// Mitsubishi GX Works2 project: PROG_ESTEIRA   PLC: Q03UDV
// PROG_ESTEIRA

PROGRAM MAIN
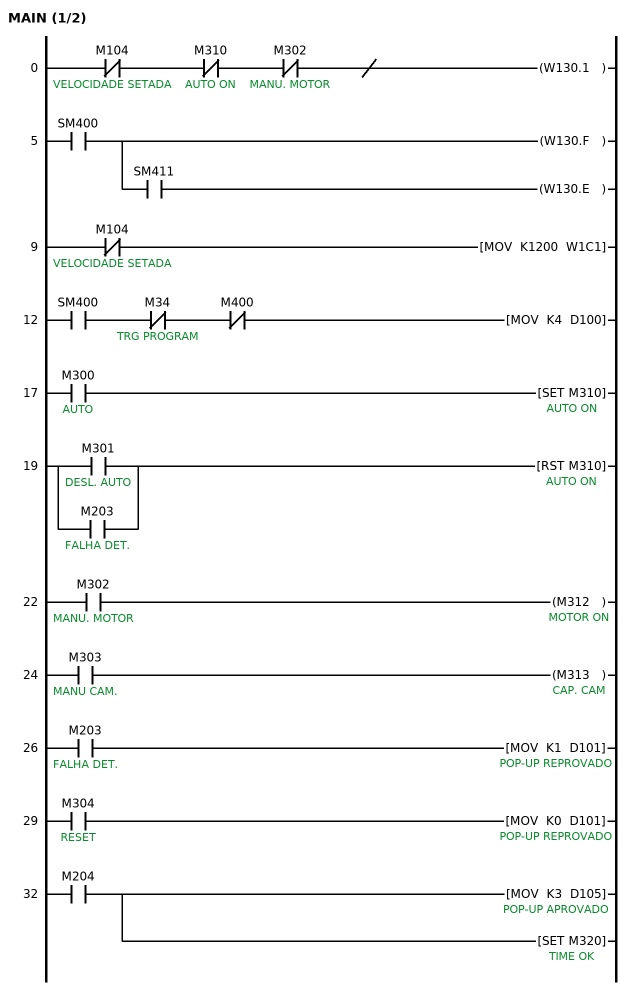
0     LDI     M104  ; VELOCIDADE SETADA
      ANI     M310  ; AUTO ON
      ANI     M302  ; MANU. MOTOR
      INV
      OUT     W130.1
5     LD      SM400
      OUT     W130.F
      AND     SM411
      OUT     W130.E
9     LDI     M104  ; VELOCIDADE SETADA
      MOV     K1200 W1C1
12    LD      SM400
      ANI     M34  ; TRG PROGRAM
      ANI     M400
      MOV     K4 D100
17    LD      M300  ; AUTO
      SET     M310  ; AUTO ON
19    LD      M301  ; DESL. AUTO
      OR      M203  ; FALHA DET.
      RST     M310  ; AUTO ON
22    LD      M302  ; MANU. MOTOR
      OUT     M312  ; MOTOR ON
24    LD      M303  ; MANU CAM.
      OUT     M313  ; CAP. CAM
26    LD      M203  ; FALHA DET.
      MOV     K1 D101  ; POP-UP REPROVADO
29    LD      M304  ; RESET
      MOV     K0 D101
32    LD      M204
      MOV     K3 D105  ; POP-UP APROVADO
      SET     M320  ; TIME OK
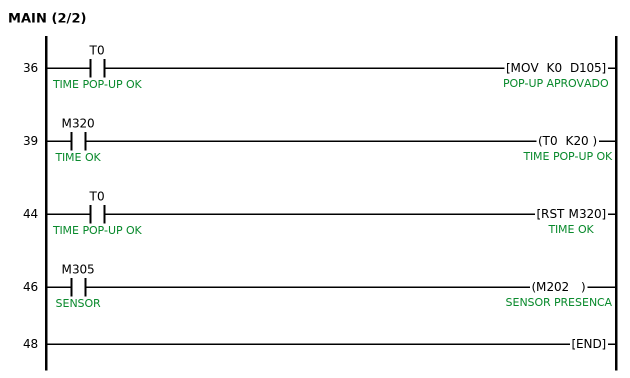
36    LD      T0  ; TIME POP-UP OK
      MOV     K0 D105
39    LD      M320  ; TIME OK
      OUT     T0 K20  ; TIME POP-UP OK
44    LD      T0  ; TIME POP-UP OK
      RST     M320  ; TIME OK
46    LD      M305  ; SENSOR
      OUT     M202  ; SENSOR PRESENCA
48    END
END_PROGRAM

// device comments not shown above
X0  ; SENSOR TRIG
M3  ; Habilitado
M36  ; NG
M100  ; Ligar
M101  ; Liga Slow Speed
M102  ; Liga Mid Speed
M103  ; Liga HIGH SPEED
M250  ; LIGA
M1000  ; LIGA
M1500  ; TEMPO PARADO AZUL
M1501  ; TEMPO PARADO VERMELHO
